FUNCTION "A-Outputs_valves" : Void
TITLE = Output_valves
{ S7_Optimized_Access := 'TRUE' }
AUTHOR : PiotrSlezak
FAMILY : Vorster
VERSION : 0.1
//Funkcja sterująca mechanizmami. Diagnostyka czujników, luzowanie, obsługa hamulca i wizualizacja stanów
   VAR_TEMP
      dummy : Bool;
      brake : Bool;
   END_VAR


BEGIN
NETWORK
TITLE = [1] GN BLOKADA_SRUBY_LEWY - HP
//[1] GN SCREW_LOCK_LEFT - HP
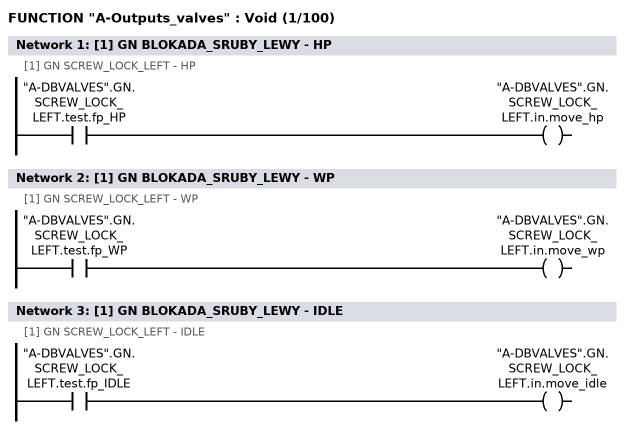
      O "A-DBVALVES".GN.SCREW_LOCK_LEFT.test.fp_HP;
//    O     "A-Flags".STATION.IN_HP_STEP
      = "A-DBVALVES".GN.SCREW_LOCK_LEFT.in.move_hp;
NETWORK
TITLE = [1] GN BLOKADA_SRUBY_LEWY - WP
//[1] GN SCREW_LOCK_LEFT - WP
      O "A-DBVALVES".GN.SCREW_LOCK_LEFT.test.fp_WP;
      = "A-DBVALVES".GN.SCREW_LOCK_LEFT.in.move_wp;
NETWORK
TITLE = [1] GN BLOKADA_SRUBY_LEWY - IDLE
//[1] GN SCREW_LOCK_LEFT - IDLE
      O "A-DBVALVES".GN.SCREW_LOCK_LEFT.test.fp_IDLE;
      = "A-DBVALVES".GN.SCREW_LOCK_LEFT.in.move_idle;
NETWORK
TITLE = [1] GN BLOKADA_SRUBY_LEWY
//[1] GN SCREW_LOCK_LEFT
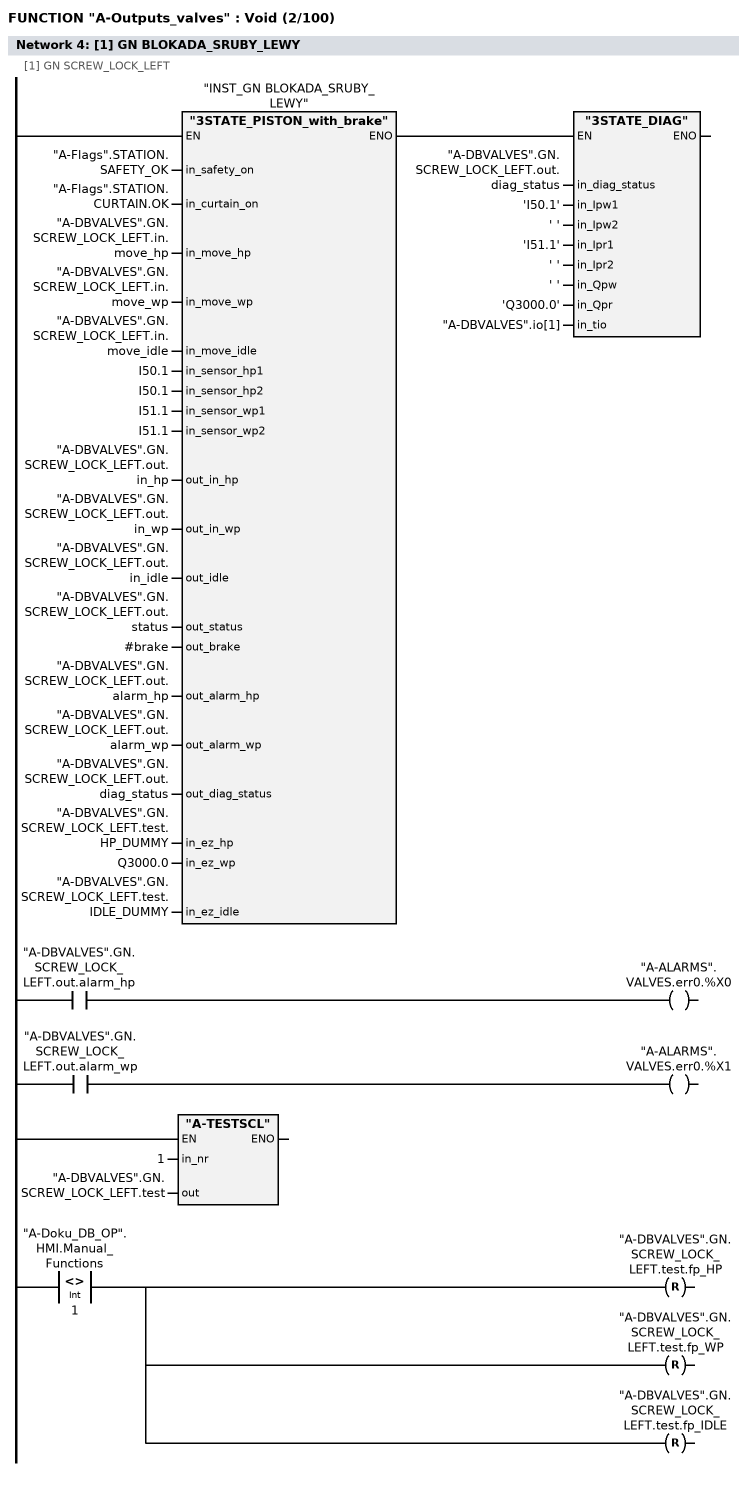
      CALL "3STATE_PISTON_with_brake", "INST_GN BLOKADA_SRUBY_LEWY"
      (  in_safety_on                := "A-Flags".STATION.SAFETY_OK ,
         in_curtain_on               := "A-Flags".STATION.CURTAIN.OK ,
         in_move_hp                  := "A-DBVALVES".GN.SCREW_LOCK_LEFT.in.move_hp ,
         in_move_wp                  := "A-DBVALVES".GN.SCREW_LOCK_LEFT.in.move_wp ,
         in_move_idle                := "A-DBVALVES".GN.SCREW_LOCK_LEFT.in.move_idle ,
         in_sensor_hp1               := I50.1 ,
         in_sensor_hp2               := I50.1 ,
         in_sensor_wp1               := I51.1 ,
         in_sensor_wp2               := I51.1 ,
         out_in_hp                   := "A-DBVALVES".GN.SCREW_LOCK_LEFT.out.in_hp ,
         out_in_wp                   := "A-DBVALVES".GN.SCREW_LOCK_LEFT.out.in_wp ,
         out_idle                    := "A-DBVALVES".GN.SCREW_LOCK_LEFT.out.in_idle ,
         out_status                  := "A-DBVALVES".GN.SCREW_LOCK_LEFT.out.status ,
         out_brake                   := #brake ,
         out_alarm_hp                := "A-DBVALVES".GN.SCREW_LOCK_LEFT.out.alarm_hp ,
         out_alarm_wp                := "A-DBVALVES".GN.SCREW_LOCK_LEFT.out.alarm_wp ,
         out_diag_status             := "A-DBVALVES".GN.SCREW_LOCK_LEFT.out.diag_status ,
         in_ez_hp                    := "A-DBVALVES".GN.SCREW_LOCK_LEFT.test.HP_DUMMY ,
         in_ez_wp                    := Q3000.0 ,
         in_ez_idle                  := "A-DBVALVES".GN.SCREW_LOCK_LEFT.test.IDLE_DUMMY
      );

      CALL "3STATE_DIAG"
      (  in_diag_status              := "A-DBVALVES".GN.SCREW_LOCK_LEFT.out.diag_status ,
         in_Ipw1                     := 'I50.1' ,
         in_Ipw2                     := ' ' ,
         in_Ipr1                     := 'I51.1' ,
         in_Ipr2                     := ' ' ,
         in_Qpw                      := ' ' ,
         in_Qpr                      := 'Q3000.0' ,
         in_tio                      := "A-DBVALVES".io[1]
      );

      A "A-DBVALVES".GN.SCREW_LOCK_LEFT.out.alarm_hp;
      = "A-ALARMS".VALVES.err0.%X0;

      A "A-DBVALVES".GN.SCREW_LOCK_LEFT.out.alarm_wp;
      = "A-ALARMS".VALVES.err0.%X1;

      CALL "A-TESTSCL"
      (  in_nr                       := 1 ,
         out                         := "A-DBVALVES".GN.SCREW_LOCK_LEFT.test
      );

      A(;
      L "A-Doku_DB_OP".HMI.Manual_Functions;
      L 1;
      <>I;
      );
      R "A-DBVALVES".GN.SCREW_LOCK_LEFT.test.fp_HP;
      R "A-DBVALVES".GN.SCREW_LOCK_LEFT.test.fp_WP;
      R "A-DBVALVES".GN.SCREW_LOCK_LEFT.test.fp_IDLE;
NETWORK
TITLE = -

NETWORK
TITLE = [2] GN BLOKADA_SRUBY_SRODEK - HP
//[2] GN SCREW_LOCK_MIDDLE - HP
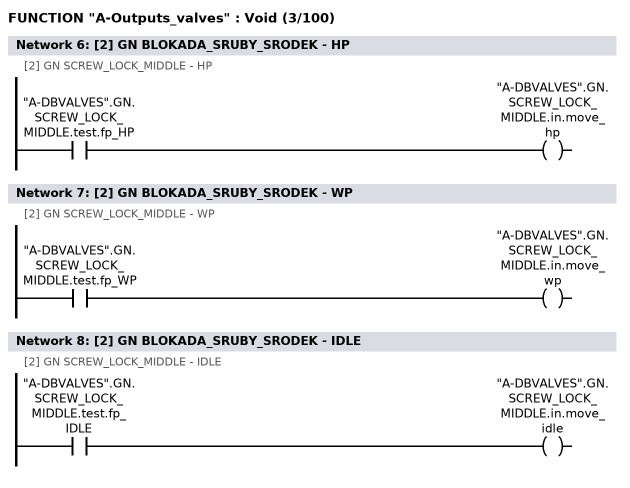
      O "A-DBVALVES".GN.SCREW_LOCK_MIDDLE.test.fp_HP;
//    O     "A-Flags".STATION.IN_HP_STEP
      = "A-DBVALVES".GN.SCREW_LOCK_MIDDLE.in.move_hp;
NETWORK
TITLE = [2] GN BLOKADA_SRUBY_SRODEK - WP
//[2] GN SCREW_LOCK_MIDDLE - WP
      O "A-DBVALVES".GN.SCREW_LOCK_MIDDLE.test.fp_WP;
      = "A-DBVALVES".GN.SCREW_LOCK_MIDDLE.in.move_wp;
NETWORK
TITLE = [2] GN BLOKADA_SRUBY_SRODEK - IDLE
//[2] GN SCREW_LOCK_MIDDLE - IDLE
      O "A-DBVALVES".GN.SCREW_LOCK_MIDDLE.test.fp_IDLE;
      = "A-DBVALVES".GN.SCREW_LOCK_MIDDLE.in.move_idle;
NETWORK
TITLE = [2] GN BLOKADA_SRUBY_SRODEK
//[2] GN SCREW_LOCK_MIDDLE
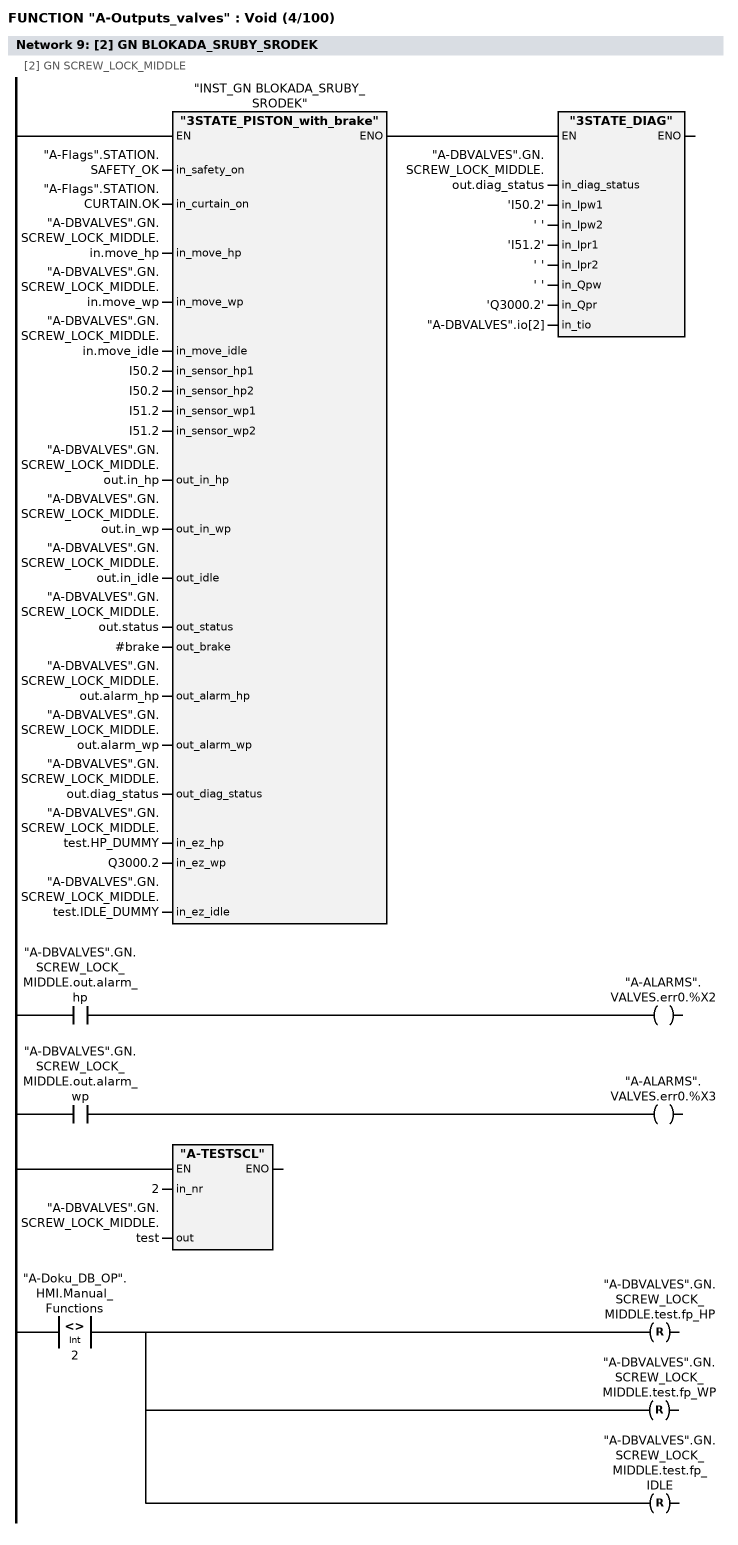
      CALL "3STATE_PISTON_with_brake", "INST_GN BLOKADA_SRUBY_SRODEK"
      (  in_safety_on                := "A-Flags".STATION.SAFETY_OK ,
         in_curtain_on               := "A-Flags".STATION.CURTAIN.OK ,
         in_move_hp                  := "A-DBVALVES".GN.SCREW_LOCK_MIDDLE.in.move_hp ,
         in_move_wp                  := "A-DBVALVES".GN.SCREW_LOCK_MIDDLE.in.move_wp ,
         in_move_idle                := "A-DBVALVES".GN.SCREW_LOCK_MIDDLE.in.move_idle ,
         in_sensor_hp1               := I50.2 ,
         in_sensor_hp2               := I50.2 ,
         in_sensor_wp1               := I51.2 ,
         in_sensor_wp2               := I51.2 ,
         out_in_hp                   := "A-DBVALVES".GN.SCREW_LOCK_MIDDLE.out.in_hp ,
         out_in_wp                   := "A-DBVALVES".GN.SCREW_LOCK_MIDDLE.out.in_wp ,
         out_idle                    := "A-DBVALVES".GN.SCREW_LOCK_MIDDLE.out.in_idle ,
         out_status                  := "A-DBVALVES".GN.SCREW_LOCK_MIDDLE.out.status ,
         out_brake                   := #brake ,
         out_alarm_hp                := "A-DBVALVES".GN.SCREW_LOCK_MIDDLE.out.alarm_hp ,
         out_alarm_wp                := "A-DBVALVES".GN.SCREW_LOCK_MIDDLE.out.alarm_wp ,
         out_diag_status             := "A-DBVALVES".GN.SCREW_LOCK_MIDDLE.out.diag_status ,
         in_ez_hp                    := "A-DBVALVES".GN.SCREW_LOCK_MIDDLE.test.HP_DUMMY ,
         in_ez_wp                    := Q3000.2 ,
         in_ez_idle                  := "A-DBVALVES".GN.SCREW_LOCK_MIDDLE.test.IDLE_DUMMY
      );

      CALL "3STATE_DIAG"
      (  in_diag_status              := "A-DBVALVES".GN.SCREW_LOCK_MIDDLE.out.diag_status ,
         in_Ipw1                     := 'I50.2' ,
         in_Ipw2                     := ' ' ,
         in_Ipr1                     := 'I51.2' ,
         in_Ipr2                     := ' ' ,
         in_Qpw                      := ' ' ,
         in_Qpr                      := 'Q3000.2' ,
         in_tio                      := "A-DBVALVES".io[2]
      );

      A "A-DBVALVES".GN.SCREW_LOCK_MIDDLE.out.alarm_hp;
      = "A-ALARMS".VALVES.err0.%X2;

      A "A-DBVALVES".GN.SCREW_LOCK_MIDDLE.out.alarm_wp;
      = "A-ALARMS".VALVES.err0.%X3;

      CALL "A-TESTSCL"
      (  in_nr                       := 2 ,
         out                         := "A-DBVALVES".GN.SCREW_LOCK_MIDDLE.test
      );

      A(;
      L "A-Doku_DB_OP".HMI.Manual_Functions;
      L 2;
      <>I;
      );
      R "A-DBVALVES".GN.SCREW_LOCK_MIDDLE.test.fp_HP;
      R "A-DBVALVES".GN.SCREW_LOCK_MIDDLE.test.fp_WP;
      R "A-DBVALVES".GN.SCREW_LOCK_MIDDLE.test.fp_IDLE;
NETWORK
TITLE = -

NETWORK
TITLE = [3] GN BLOKADA_SRUBY_PRAWY - HP
//[3] GN SCREW_LOCK_RIGHT - HP
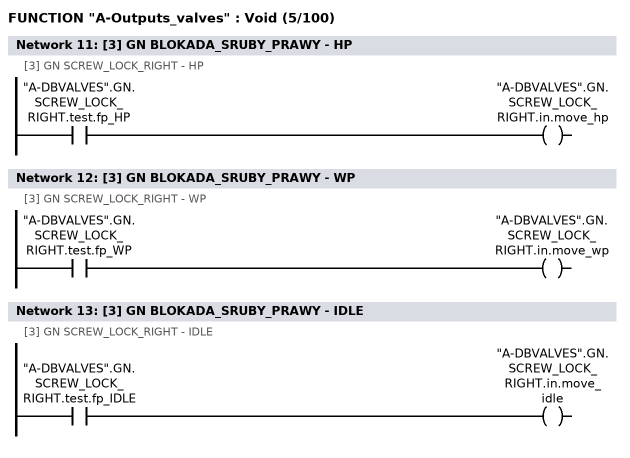
      O "A-DBVALVES".GN.SCREW_LOCK_RIGHT.test.fp_HP;
//    O     "A-Flags".STATION.IN_HP_STEP
      = "A-DBVALVES".GN.SCREW_LOCK_RIGHT.in.move_hp;
NETWORK
TITLE = [3] GN BLOKADA_SRUBY_PRAWY - WP
//[3] GN SCREW_LOCK_RIGHT - WP
      O "A-DBVALVES".GN.SCREW_LOCK_RIGHT.test.fp_WP;
      = "A-DBVALVES".GN.SCREW_LOCK_RIGHT.in.move_wp;
NETWORK
TITLE = [3] GN BLOKADA_SRUBY_PRAWY - IDLE
//[3] GN SCREW_LOCK_RIGHT - IDLE
      O "A-DBVALVES".GN.SCREW_LOCK_RIGHT.test.fp_IDLE;
      = "A-DBVALVES".GN.SCREW_LOCK_RIGHT.in.move_idle;
NETWORK
TITLE = [3] GN BLOKADA_SRUBY_PRAWY
//[3] GN SCREW_LOCK_RIGHT
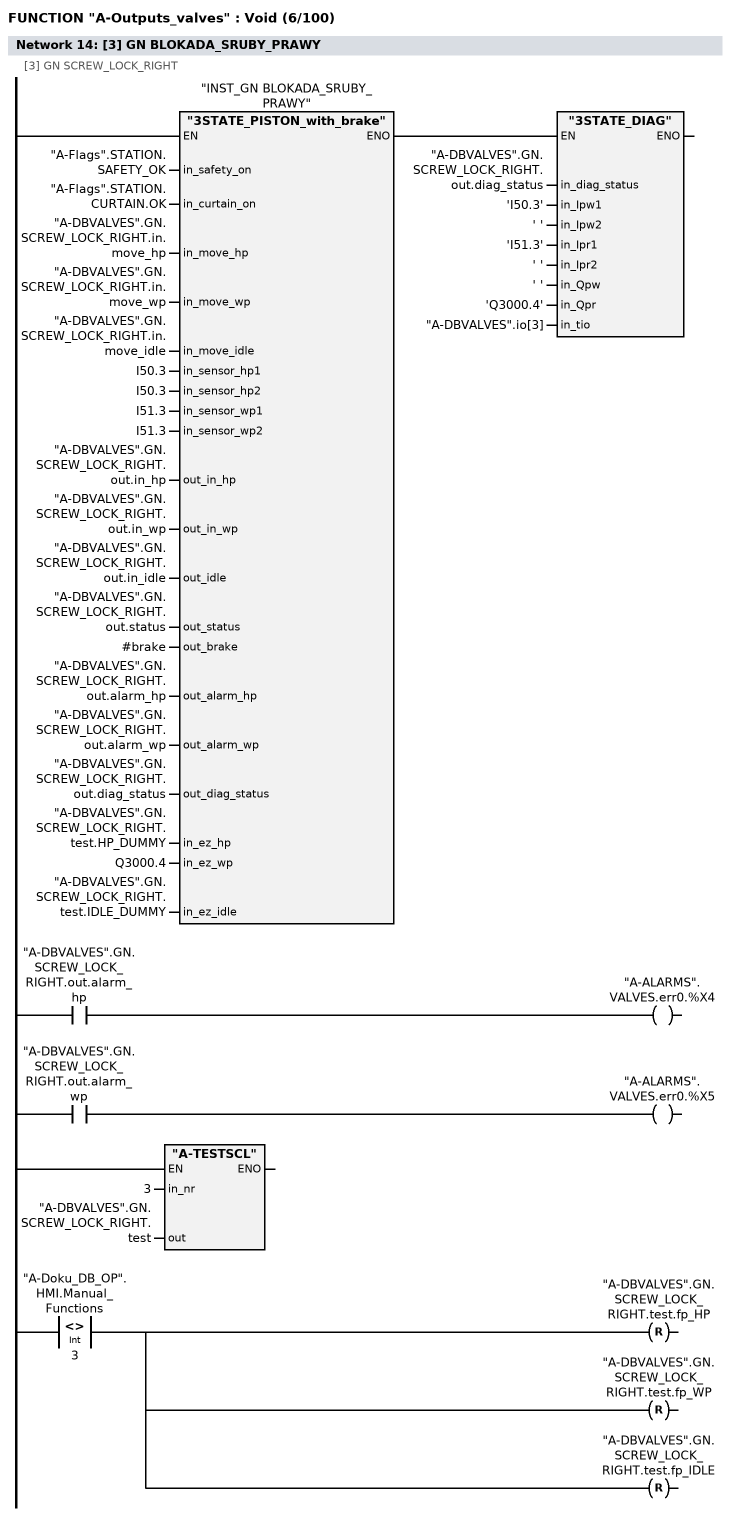
      CALL "3STATE_PISTON_with_brake", "INST_GN BLOKADA_SRUBY_PRAWY"
      (  in_safety_on                := "A-Flags".STATION.SAFETY_OK ,
         in_curtain_on               := "A-Flags".STATION.CURTAIN.OK ,
         in_move_hp                  := "A-DBVALVES".GN.SCREW_LOCK_RIGHT.in.move_hp ,
         in_move_wp                  := "A-DBVALVES".GN.SCREW_LOCK_RIGHT.in.move_wp ,
         in_move_idle                := "A-DBVALVES".GN.SCREW_LOCK_RIGHT.in.move_idle ,
         in_sensor_hp1               := I50.3 ,
         in_sensor_hp2               := I50.3 ,
         in_sensor_wp1               := I51.3 ,
         in_sensor_wp2               := I51.3 ,
         out_in_hp                   := "A-DBVALVES".GN.SCREW_LOCK_RIGHT.out.in_hp ,
         out_in_wp                   := "A-DBVALVES".GN.SCREW_LOCK_RIGHT.out.in_wp ,
         out_idle                    := "A-DBVALVES".GN.SCREW_LOCK_RIGHT.out.in_idle ,
         out_status                  := "A-DBVALVES".GN.SCREW_LOCK_RIGHT.out.status ,
         out_brake                   := #brake ,
         out_alarm_hp                := "A-DBVALVES".GN.SCREW_LOCK_RIGHT.out.alarm_hp ,
         out_alarm_wp                := "A-DBVALVES".GN.SCREW_LOCK_RIGHT.out.alarm_wp ,
         out_diag_status             := "A-DBVALVES".GN.SCREW_LOCK_RIGHT.out.diag_status ,
         in_ez_hp                    := "A-DBVALVES".GN.SCREW_LOCK_RIGHT.test.HP_DUMMY ,
         in_ez_wp                    := Q3000.4 ,
         in_ez_idle                  := "A-DBVALVES".GN.SCREW_LOCK_RIGHT.test.IDLE_DUMMY
      );

      CALL "3STATE_DIAG"
      (  in_diag_status              := "A-DBVALVES".GN.SCREW_LOCK_RIGHT.out.diag_status ,
         in_Ipw1                     := 'I50.3' ,
         in_Ipw2                     := ' ' ,
         in_Ipr1                     := 'I51.3' ,
         in_Ipr2                     := ' ' ,
         in_Qpw                      := ' ' ,
         in_Qpr                      := 'Q3000.4' ,
         in_tio                      := "A-DBVALVES".io[3]
      );

      A "A-DBVALVES".GN.SCREW_LOCK_RIGHT.out.alarm_hp;
      = "A-ALARMS".VALVES.err0.%X4;

      A "A-DBVALVES".GN.SCREW_LOCK_RIGHT.out.alarm_wp;
      = "A-ALARMS".VALVES.err0.%X5;

      CALL "A-TESTSCL"
      (  in_nr                       := 3 ,
         out                         := "A-DBVALVES".GN.SCREW_LOCK_RIGHT.test
      );

      A(;
      L "A-Doku_DB_OP".HMI.Manual_Functions;
      L 3;
      <>I;
      );
      R "A-DBVALVES".GN.SCREW_LOCK_RIGHT.test.fp_HP;
      R "A-DBVALVES".GN.SCREW_LOCK_RIGHT.test.fp_WP;
      R "A-DBVALVES".GN.SCREW_LOCK_RIGHT.test.fp_IDLE;
NETWORK
TITLE = -

NETWORK
TITLE = [4] GN ZASUWKA - HP
//[4] GN LATCH - HP
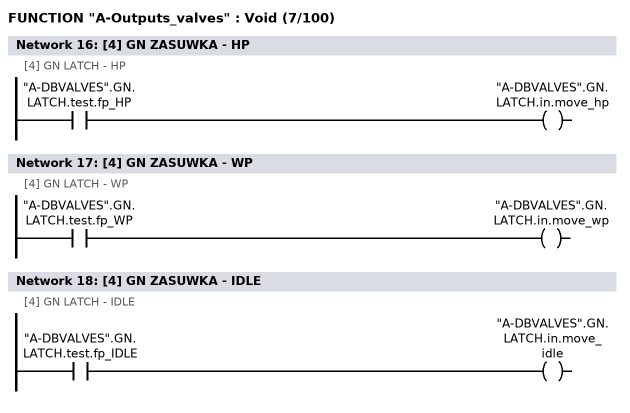
      O "A-DBVALVES".GN.LATCH.test.fp_HP;
//    O     "A-Flags".STATION.IN_HP_STEP
      = "A-DBVALVES".GN.LATCH.in.move_hp;
NETWORK
TITLE = [4] GN ZASUWKA - WP
//[4] GN LATCH - WP
      O "A-DBVALVES".GN.LATCH.test.fp_WP;
      = "A-DBVALVES".GN.LATCH.in.move_wp;
NETWORK
TITLE = [4] GN ZASUWKA - IDLE
//[4] GN LATCH - IDLE
      O "A-DBVALVES".GN.LATCH.test.fp_IDLE;
      = "A-DBVALVES".GN.LATCH.in.move_idle;
NETWORK
TITLE = [4] GN ZASUWKA
//[4] GN LATCH
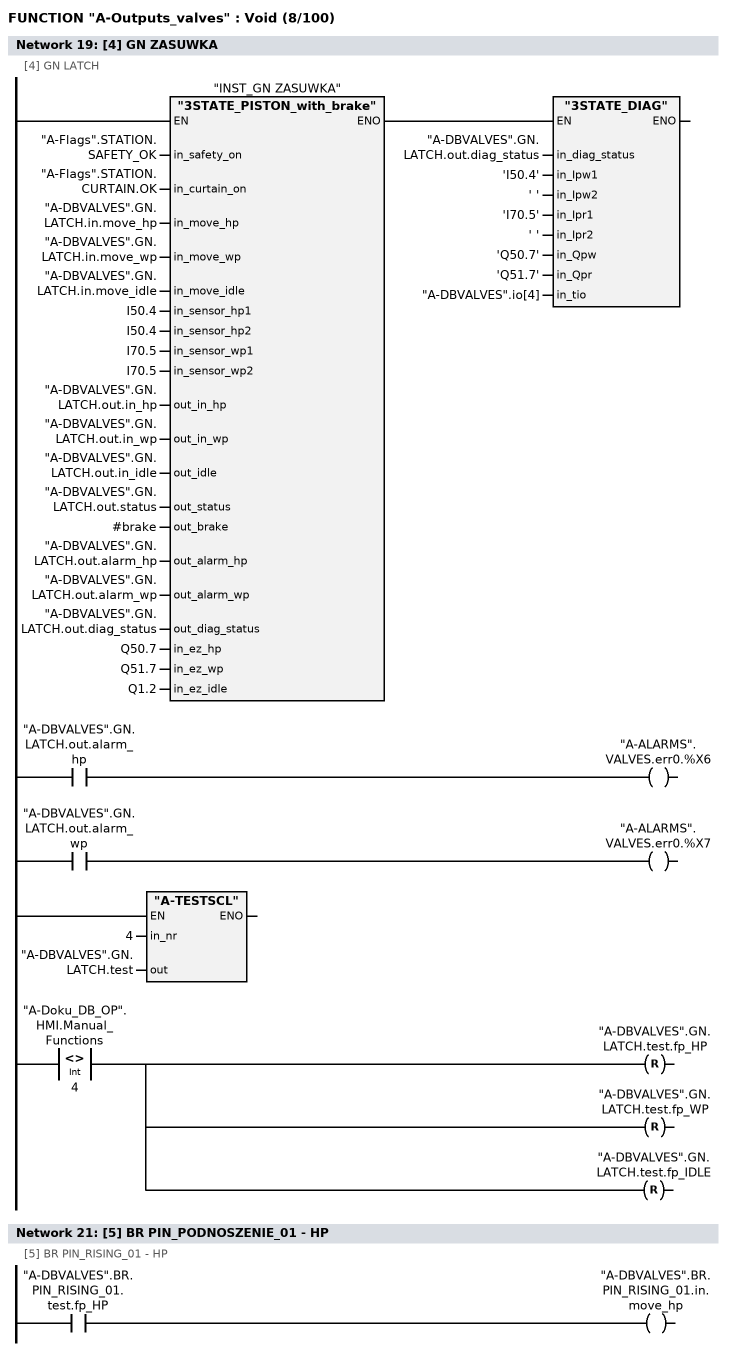
      CALL "3STATE_PISTON_with_brake", "INST_GN ZASUWKA"
      (  in_safety_on                := "A-Flags".STATION.SAFETY_OK ,
         in_curtain_on               := "A-Flags".STATION.CURTAIN.OK ,
         in_move_hp                  := "A-DBVALVES".GN.LATCH.in.move_hp ,
         in_move_wp                  := "A-DBVALVES".GN.LATCH.in.move_wp ,
         in_move_idle                := "A-DBVALVES".GN.LATCH.in.move_idle ,
         in_sensor_hp1               := I50.4 ,
         in_sensor_hp2               := I50.4 ,
         in_sensor_wp1               := I70.5 ,
         in_sensor_wp2               := I70.5 ,
         out_in_hp                   := "A-DBVALVES".GN.LATCH.out.in_hp ,
         out_in_wp                   := "A-DBVALVES".GN.LATCH.out.in_wp ,
         out_idle                    := "A-DBVALVES".GN.LATCH.out.in_idle ,
         out_status                  := "A-DBVALVES".GN.LATCH.out.status ,
         out_brake                   := #brake ,
         out_alarm_hp                := "A-DBVALVES".GN.LATCH.out.alarm_hp ,
         out_alarm_wp                := "A-DBVALVES".GN.LATCH.out.alarm_wp ,
         out_diag_status             := "A-DBVALVES".GN.LATCH.out.diag_status ,
         in_ez_hp                    := Q50.7 ,
         in_ez_wp                    := Q51.7 ,
         in_ez_idle                  := Q1.2
      );

      CALL "3STATE_DIAG"
      (  in_diag_status              := "A-DBVALVES".GN.LATCH.out.diag_status ,
         in_Ipw1                     := 'I50.4' ,
         in_Ipw2                     := ' ' ,
         in_Ipr1                     := 'I70.5' ,
         in_Ipr2                     := ' ' ,
         in_Qpw                      := 'Q50.7' ,
         in_Qpr                      := 'Q51.7' ,
         in_tio                      := "A-DBVALVES".io[4]
      );

      A "A-DBVALVES".GN.LATCH.out.alarm_hp;
      = "A-ALARMS".VALVES.err0.%X6;

      A "A-DBVALVES".GN.LATCH.out.alarm_wp;
      = "A-ALARMS".VALVES.err0.%X7;

      CALL "A-TESTSCL"
      (  in_nr                       := 4 ,
         out                         := "A-DBVALVES".GN.LATCH.test
      );

      A(;
      L "A-Doku_DB_OP".HMI.Manual_Functions;
      L 4;
      <>I;
      );
      R "A-DBVALVES".GN.LATCH.test.fp_HP;
      R "A-DBVALVES".GN.LATCH.test.fp_WP;
      R "A-DBVALVES".GN.LATCH.test.fp_IDLE;
NETWORK
TITLE = -

NETWORK
TITLE = [5] BR PIN_PODNOSZENIE_01 - HP
//[5] BR PIN_RISING_01 - HP
      O "A-DBVALVES".BR.PIN_RISING_01.test.fp_HP;
//    O     "A-Flags".STATION.IN_HP_STEP
      = "A-DBVALVES".BR.PIN_RISING_01.in.move_hp;
NETWORK
TITLE = [5] BR PIN_PODNOSZENIE_01 - WP
//[5] BR PIN_RISING_01 - WP
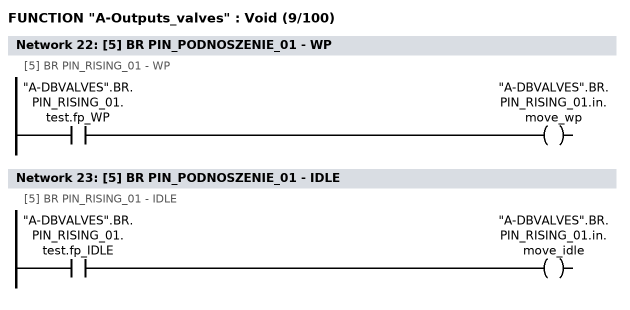
      O "A-DBVALVES".BR.PIN_RISING_01.test.fp_WP;
      = "A-DBVALVES".BR.PIN_RISING_01.in.move_wp;
NETWORK
TITLE = [5] BR PIN_PODNOSZENIE_01 - IDLE
//[5] BR PIN_RISING_01 - IDLE
      O "A-DBVALVES".BR.PIN_RISING_01.test.fp_IDLE;
      = "A-DBVALVES".BR.PIN_RISING_01.in.move_idle;
NETWORK
TITLE = [5] BR PIN_PODNOSZENIE_01
//[5] BR PIN_RISING_01
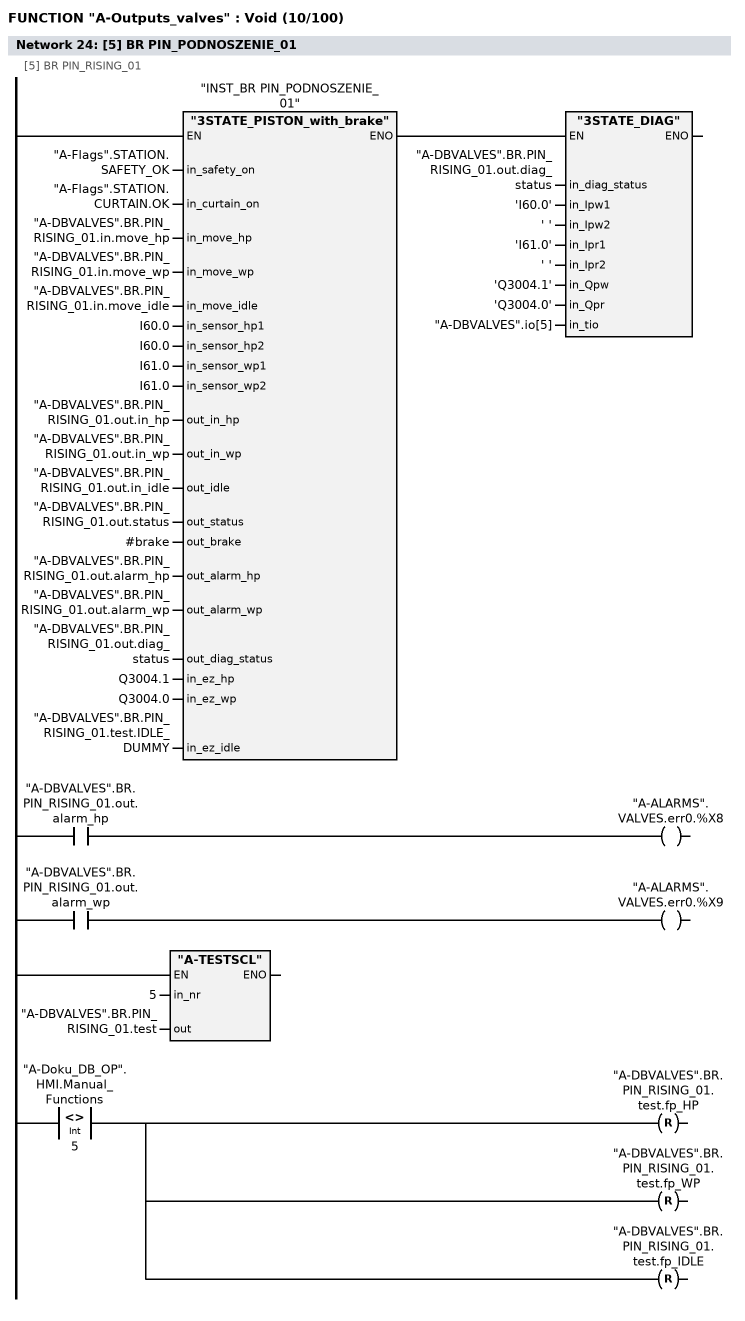
      CALL "3STATE_PISTON_with_brake", "INST_BR PIN_PODNOSZENIE_01"
      (  in_safety_on                := "A-Flags".STATION.SAFETY_OK ,
         in_curtain_on               := "A-Flags".STATION.CURTAIN.OK ,
         in_move_hp                  := "A-DBVALVES".BR.PIN_RISING_01.in.move_hp ,
         in_move_wp                  := "A-DBVALVES".BR.PIN_RISING_01.in.move_wp ,
         in_move_idle                := "A-DBVALVES".BR.PIN_RISING_01.in.move_idle ,
         in_sensor_hp1               := I60.0 ,
         in_sensor_hp2               := I60.0 ,
         in_sensor_wp1               := I61.0 ,
         in_sensor_wp2               := I61.0 ,
         out_in_hp                   := "A-DBVALVES".BR.PIN_RISING_01.out.in_hp ,
         out_in_wp                   := "A-DBVALVES".BR.PIN_RISING_01.out.in_wp ,
         out_idle                    := "A-DBVALVES".BR.PIN_RISING_01.out.in_idle ,
         out_status                  := "A-DBVALVES".BR.PIN_RISING_01.out.status ,
         out_brake                   := #brake ,
         out_alarm_hp                := "A-DBVALVES".BR.PIN_RISING_01.out.alarm_hp ,
         out_alarm_wp                := "A-DBVALVES".BR.PIN_RISING_01.out.alarm_wp ,
         out_diag_status             := "A-DBVALVES".BR.PIN_RISING_01.out.diag_status ,
         in_ez_hp                    := Q3004.1 ,
         in_ez_wp                    := Q3004.0 ,
         in_ez_idle                  := "A-DBVALVES".BR.PIN_RISING_01.test.IDLE_DUMMY
      );

      CALL "3STATE_DIAG"
      (  in_diag_status              := "A-DBVALVES".BR.PIN_RISING_01.out.diag_status ,
         in_Ipw1                     := 'I60.0' ,
         in_Ipw2                     := ' ' ,
         in_Ipr1                     := 'I61.0' ,
         in_Ipr2                     := ' ' ,
         in_Qpw                      := 'Q3004.1' ,
         in_Qpr                      := 'Q3004.0' ,
         in_tio                      := "A-DBVALVES".io[5]
      );

      A "A-DBVALVES".BR.PIN_RISING_01.out.alarm_hp;
      = "A-ALARMS".VALVES.err0.%X8;

      A "A-DBVALVES".BR.PIN_RISING_01.out.alarm_wp;
      = "A-ALARMS".VALVES.err0.%X9;

      CALL "A-TESTSCL"
      (  in_nr                       := 5 ,
         out                         := "A-DBVALVES".BR.PIN_RISING_01.test
      );

      A(;
      L "A-Doku_DB_OP".HMI.Manual_Functions;
      L 5;
      <>I;
      );
      R "A-DBVALVES".BR.PIN_RISING_01.test.fp_HP;
      R "A-DBVALVES".BR.PIN_RISING_01.test.fp_WP;
      R "A-DBVALVES".BR.PIN_RISING_01.test.fp_IDLE;
NETWORK
TITLE = -

NETWORK
TITLE = [6] BR PIN_01 - HP
//[6] BR PIN_01 - HP
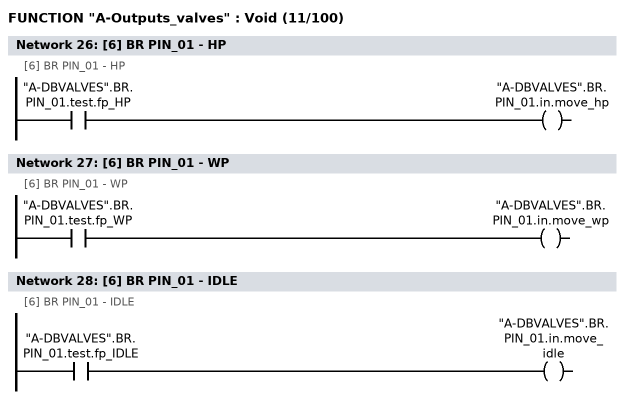
      O "A-DBVALVES".BR.PIN_01.test.fp_HP;
//    O     "A-Flags".STATION.IN_HP_STEP
      = "A-DBVALVES".BR.PIN_01.in.move_hp;
NETWORK
TITLE = [6] BR PIN_01 - WP
//[6] BR PIN_01 - WP
      O "A-DBVALVES".BR.PIN_01.test.fp_WP;
      = "A-DBVALVES".BR.PIN_01.in.move_wp;
NETWORK
TITLE = [6] BR PIN_01 - IDLE
//[6] BR PIN_01 - IDLE
      O "A-DBVALVES".BR.PIN_01.test.fp_IDLE;
      = "A-DBVALVES".BR.PIN_01.in.move_idle;
NETWORK
TITLE = [6] BR PIN_01
//[6] BR PIN_01
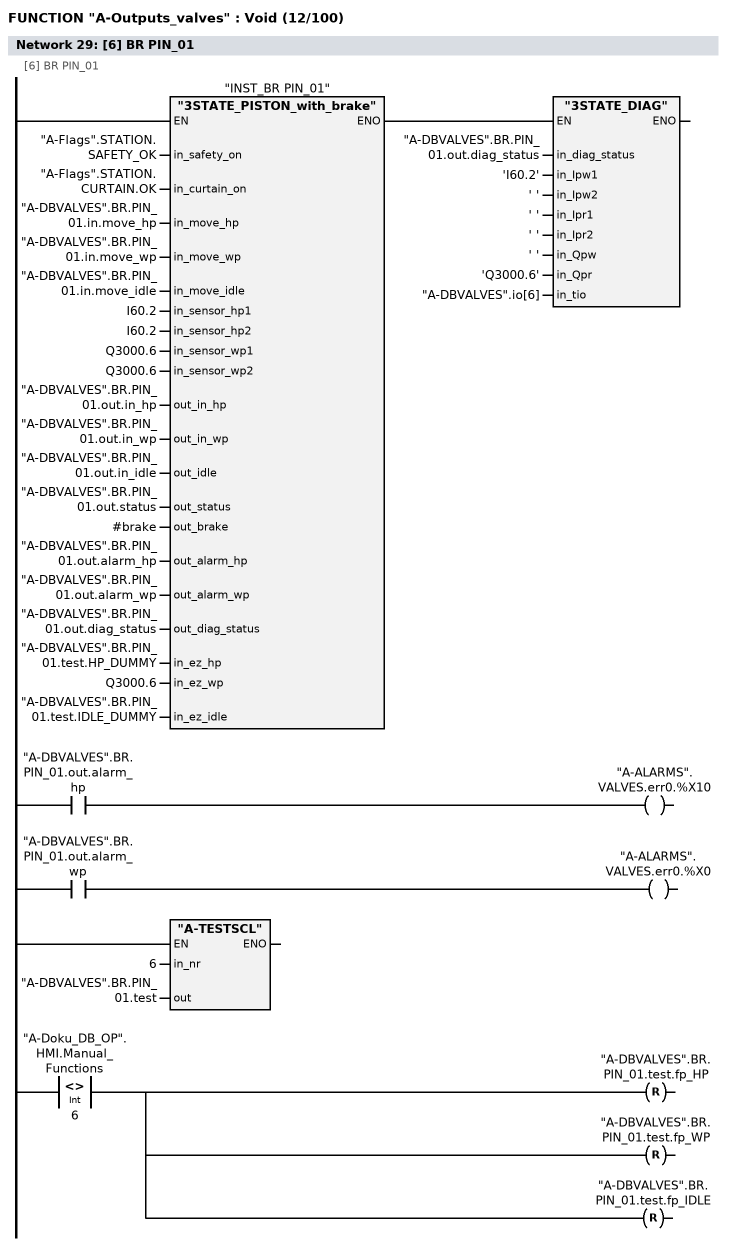
      CALL "3STATE_PISTON_with_brake", "INST_BR PIN_01"
      (  in_safety_on                := "A-Flags".STATION.SAFETY_OK ,
         in_curtain_on               := "A-Flags".STATION.CURTAIN.OK ,
         in_move_hp                  := "A-DBVALVES".BR.PIN_01.in.move_hp ,
         in_move_wp                  := "A-DBVALVES".BR.PIN_01.in.move_wp ,
         in_move_idle                := "A-DBVALVES".BR.PIN_01.in.move_idle ,
         in_sensor_hp1               := I60.2 ,
         in_sensor_hp2               := I60.2 ,
         in_sensor_wp1               := Q3000.6 ,
         in_sensor_wp2               := Q3000.6 ,
         out_in_hp                   := "A-DBVALVES".BR.PIN_01.out.in_hp ,
         out_in_wp                   := "A-DBVALVES".BR.PIN_01.out.in_wp ,
         out_idle                    := "A-DBVALVES".BR.PIN_01.out.in_idle ,
         out_status                  := "A-DBVALVES".BR.PIN_01.out.status ,
         out_brake                   := #brake ,
         out_alarm_hp                := "A-DBVALVES".BR.PIN_01.out.alarm_hp ,
         out_alarm_wp                := "A-DBVALVES".BR.PIN_01.out.alarm_wp ,
         out_diag_status             := "A-DBVALVES".BR.PIN_01.out.diag_status ,
         in_ez_hp                    := "A-DBVALVES".BR.PIN_01.test.HP_DUMMY ,
         in_ez_wp                    := Q3000.6 ,
         in_ez_idle                  := "A-DBVALVES".BR.PIN_01.test.IDLE_DUMMY
      );

      CALL "3STATE_DIAG"
      (  in_diag_status              := "A-DBVALVES".BR.PIN_01.out.diag_status ,
         in_Ipw1                     := 'I60.2' ,
         in_Ipw2                     := ' ' ,
         in_Ipr1                     := ' ' ,
         in_Ipr2                     := ' ' ,
         in_Qpw                      := ' ' ,
         in_Qpr                      := 'Q3000.6' ,
         in_tio                      := "A-DBVALVES".io[6]
      );

      A "A-DBVALVES".BR.PIN_01.out.alarm_hp;
      = "A-ALARMS".VALVES.err0.%X10;

      A "A-DBVALVES".BR.PIN_01.out.alarm_wp;
      = "A-ALARMS".VALVES.err0.%X0;

      CALL "A-TESTSCL"
      (  in_nr                       := 6 ,
         out                         := "A-DBVALVES".BR.PIN_01.test
      );

      A(;
      L "A-Doku_DB_OP".HMI.Manual_Functions;
      L 6;
      <>I;
      );
      R "A-DBVALVES".BR.PIN_01.test.fp_HP;
      R "A-DBVALVES".BR.PIN_01.test.fp_WP;
      R "A-DBVALVES".BR.PIN_01.test.fp_IDLE;
NETWORK
TITLE = -

NETWORK
TITLE = [7] BR PIN_PODNOSZENIE_02 - HP
//[7] BR PIN_RISING_02 - HP
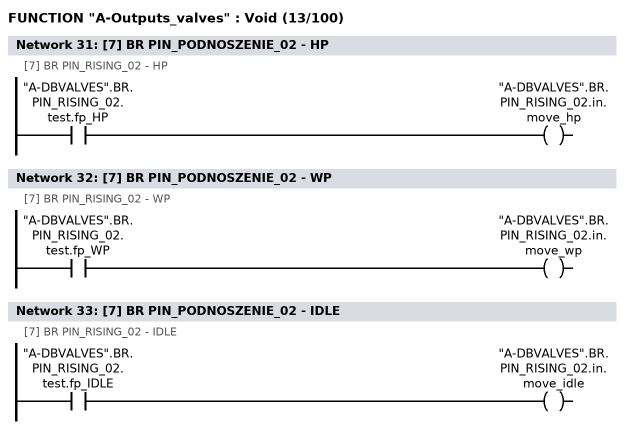
      O "A-DBVALVES".BR.PIN_RISING_02.test.fp_HP;
//    O     "A-Flags".STATION.IN_HP_STEP
      = "A-DBVALVES".BR.PIN_RISING_02.in.move_hp;
NETWORK
TITLE = [7] BR PIN_PODNOSZENIE_02 - WP
//[7] BR PIN_RISING_02 - WP
      O "A-DBVALVES".BR.PIN_RISING_02.test.fp_WP;
      = "A-DBVALVES".BR.PIN_RISING_02.in.move_wp;
NETWORK
TITLE = [7] BR PIN_PODNOSZENIE_02 - IDLE
//[7] BR PIN_RISING_02 - IDLE
      O "A-DBVALVES".BR.PIN_RISING_02.test.fp_IDLE;
      = "A-DBVALVES".BR.PIN_RISING_02.in.move_idle;
NETWORK
TITLE = [7] BR PIN_PODNOSZENIE_02
//[7] BR PIN_RISING_02
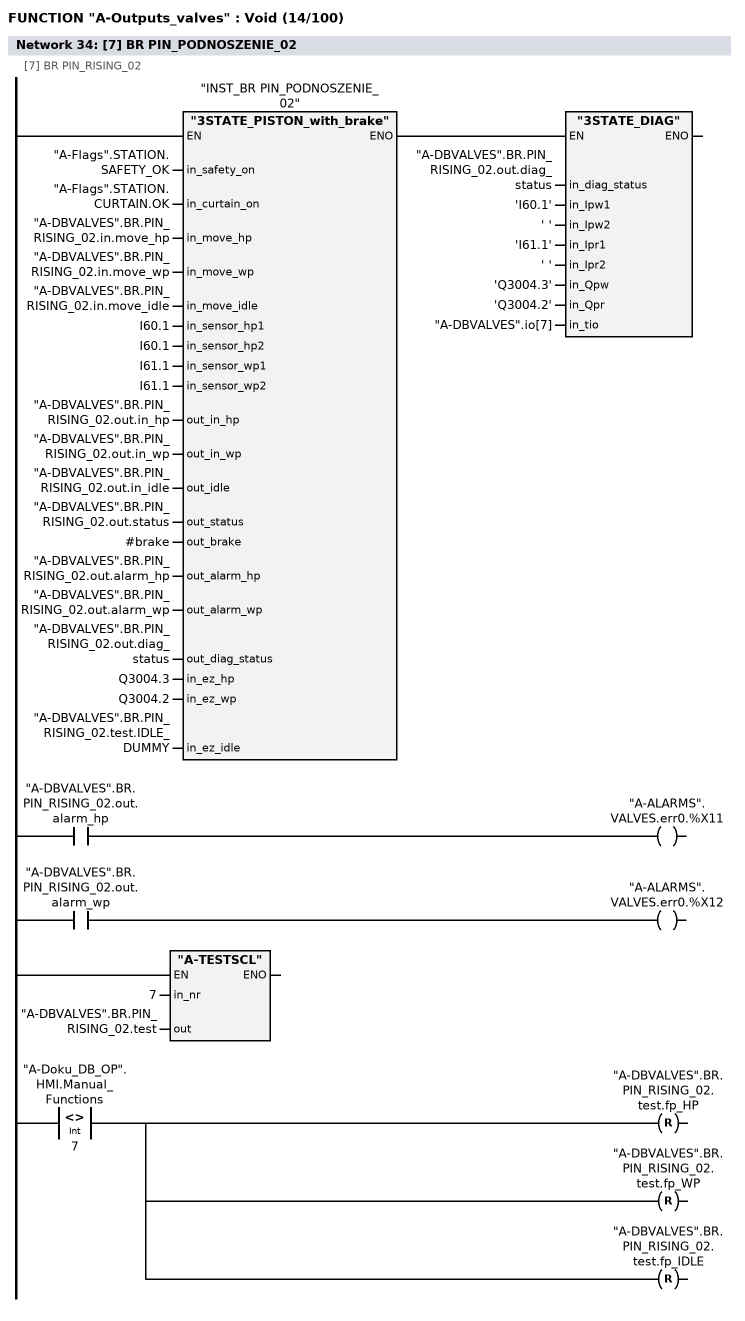
      CALL "3STATE_PISTON_with_brake", "INST_BR PIN_PODNOSZENIE_02"
      (  in_safety_on                := "A-Flags".STATION.SAFETY_OK ,
         in_curtain_on               := "A-Flags".STATION.CURTAIN.OK ,
         in_move_hp                  := "A-DBVALVES".BR.PIN_RISING_02.in.move_hp ,
         in_move_wp                  := "A-DBVALVES".BR.PIN_RISING_02.in.move_wp ,
         in_move_idle                := "A-DBVALVES".BR.PIN_RISING_02.in.move_idle ,
         in_sensor_hp1               := I60.1 ,
         in_sensor_hp2               := I60.1 ,
         in_sensor_wp1               := I61.1 ,
         in_sensor_wp2               := I61.1 ,
         out_in_hp                   := "A-DBVALVES".BR.PIN_RISING_02.out.in_hp ,
         out_in_wp                   := "A-DBVALVES".BR.PIN_RISING_02.out.in_wp ,
         out_idle                    := "A-DBVALVES".BR.PIN_RISING_02.out.in_idle ,
         out_status                  := "A-DBVALVES".BR.PIN_RISING_02.out.status ,
         out_brake                   := #brake ,
         out_alarm_hp                := "A-DBVALVES".BR.PIN_RISING_02.out.alarm_hp ,
         out_alarm_wp                := "A-DBVALVES".BR.PIN_RISING_02.out.alarm_wp ,
         out_diag_status             := "A-DBVALVES".BR.PIN_RISING_02.out.diag_status ,
         in_ez_hp                    := Q3004.3 ,
         in_ez_wp                    := Q3004.2 ,
         in_ez_idle                  := "A-DBVALVES".BR.PIN_RISING_02.test.IDLE_DUMMY
      );

      CALL "3STATE_DIAG"
      (  in_diag_status              := "A-DBVALVES".BR.PIN_RISING_02.out.diag_status ,
         in_Ipw1                     := 'I60.1' ,
         in_Ipw2                     := ' ' ,
         in_Ipr1                     := 'I61.1' ,
         in_Ipr2                     := ' ' ,
         in_Qpw                      := 'Q3004.3' ,
         in_Qpr                      := 'Q3004.2' ,
         in_tio                      := "A-DBVALVES".io[7]
      );

      A "A-DBVALVES".BR.PIN_RISING_02.out.alarm_hp;
      = "A-ALARMS".VALVES.err0.%X11;

      A "A-DBVALVES".BR.PIN_RISING_02.out.alarm_wp;
      = "A-ALARMS".VALVES.err0.%X12;

      CALL "A-TESTSCL"
      (  in_nr                       := 7 ,
         out                         := "A-DBVALVES".BR.PIN_RISING_02.test
      );

      A(;
      L "A-Doku_DB_OP".HMI.Manual_Functions;
      L 7;
      <>I;
      );
      R "A-DBVALVES".BR.PIN_RISING_02.test.fp_HP;
      R "A-DBVALVES".BR.PIN_RISING_02.test.fp_WP;
      R "A-DBVALVES".BR.PIN_RISING_02.test.fp_IDLE;
NETWORK
TITLE = -

NETWORK
TITLE = [8] BR PIN_02 - HP
//[8] BR PIN_02 - HP
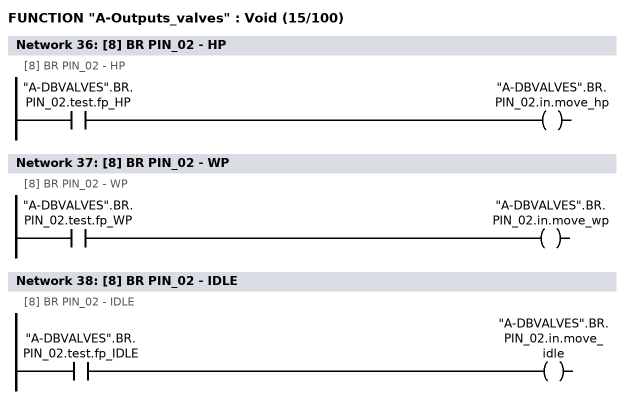
      O "A-DBVALVES".BR.PIN_02.test.fp_HP;
//    O     "A-Flags".STATION.IN_HP_STEP
      = "A-DBVALVES".BR.PIN_02.in.move_hp;
NETWORK
TITLE = [8] BR PIN_02 - WP
//[8] BR PIN_02 - WP
      O "A-DBVALVES".BR.PIN_02.test.fp_WP;
      = "A-DBVALVES".BR.PIN_02.in.move_wp;
NETWORK
TITLE = [8] BR PIN_02 - IDLE
//[8] BR PIN_02 - IDLE
      O "A-DBVALVES".BR.PIN_02.test.fp_IDLE;
      = "A-DBVALVES".BR.PIN_02.in.move_idle;
NETWORK
TITLE = [8] BR PIN_02
//[8] BR PIN_02
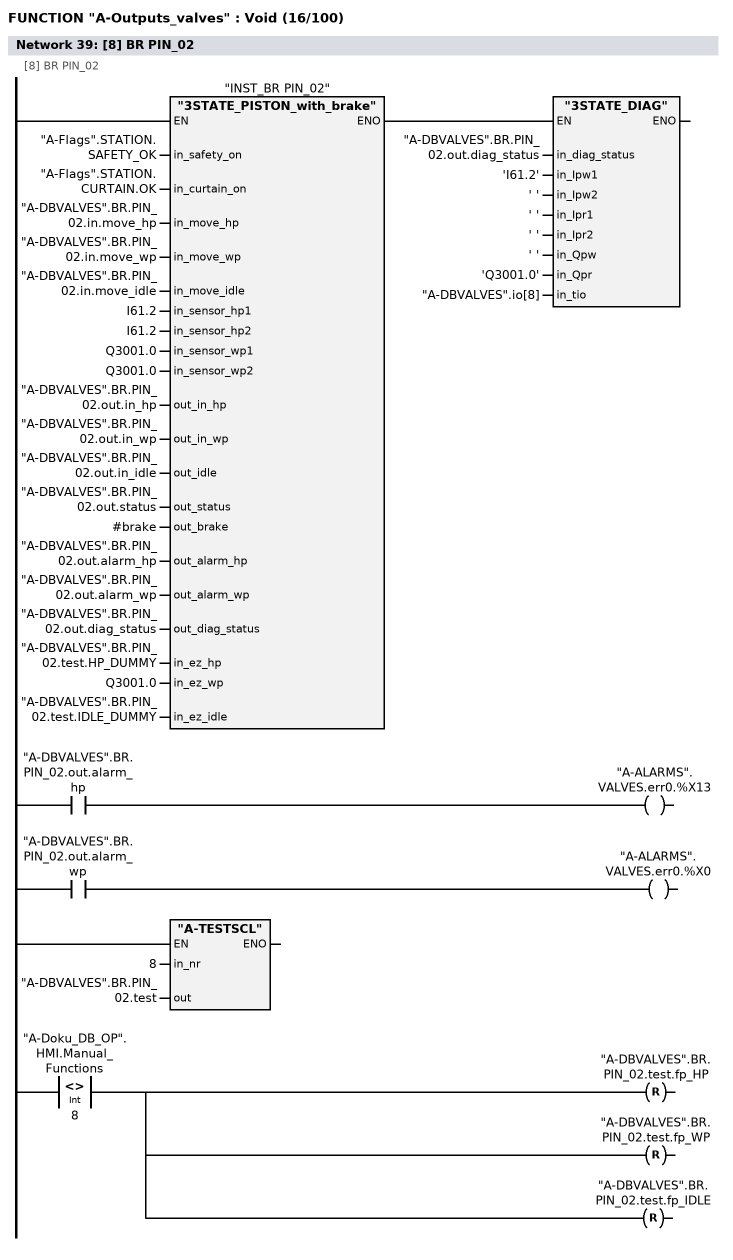
      CALL "3STATE_PISTON_with_brake", "INST_BR PIN_02"
      (  in_safety_on                := "A-Flags".STATION.SAFETY_OK ,
         in_curtain_on               := "A-Flags".STATION.CURTAIN.OK ,
         in_move_hp                  := "A-DBVALVES".BR.PIN_02.in.move_hp ,
         in_move_wp                  := "A-DBVALVES".BR.PIN_02.in.move_wp ,
         in_move_idle                := "A-DBVALVES".BR.PIN_02.in.move_idle ,
         in_sensor_hp1               := I61.2 ,
         in_sensor_hp2               := I61.2 ,
         in_sensor_wp1               := Q3001.0 ,
         in_sensor_wp2               := Q3001.0 ,
         out_in_hp                   := "A-DBVALVES".BR.PIN_02.out.in_hp ,
         out_in_wp                   := "A-DBVALVES".BR.PIN_02.out.in_wp ,
         out_idle                    := "A-DBVALVES".BR.PIN_02.out.in_idle ,
         out_status                  := "A-DBVALVES".BR.PIN_02.out.status ,
         out_brake                   := #brake ,
         out_alarm_hp                := "A-DBVALVES".BR.PIN_02.out.alarm_hp ,
         out_alarm_wp                := "A-DBVALVES".BR.PIN_02.out.alarm_wp ,
         out_diag_status             := "A-DBVALVES".BR.PIN_02.out.diag_status ,
         in_ez_hp                    := "A-DBVALVES".BR.PIN_02.test.HP_DUMMY ,
         in_ez_wp                    := Q3001.0 ,
         in_ez_idle                  := "A-DBVALVES".BR.PIN_02.test.IDLE_DUMMY
      );

      CALL "3STATE_DIAG"
      (  in_diag_status              := "A-DBVALVES".BR.PIN_02.out.diag_status ,
         in_Ipw1                     := 'I61.2' ,
         in_Ipw2                     := ' ' ,
         in_Ipr1                     := ' ' ,
         in_Ipr2                     := ' ' ,
         in_Qpw                      := ' ' ,
         in_Qpr                      := 'Q3001.0' ,
         in_tio                      := "A-DBVALVES".io[8]
      );

      A "A-DBVALVES".BR.PIN_02.out.alarm_hp;
      = "A-ALARMS".VALVES.err0.%X13;

      A "A-DBVALVES".BR.PIN_02.out.alarm_wp;
      = "A-ALARMS".VALVES.err0.%X0;

      CALL "A-TESTSCL"
      (  in_nr                       := 8 ,
         out                         := "A-DBVALVES".BR.PIN_02.test
      );

      A(;
      L "A-Doku_DB_OP".HMI.Manual_Functions;
      L 8;
      <>I;
      );
      R "A-DBVALVES".BR.PIN_02.test.fp_HP;
      R "A-DBVALVES".BR.PIN_02.test.fp_WP;
      R "A-DBVALVES".BR.PIN_02.test.fp_IDLE;
NETWORK
TITLE = -

NETWORK
TITLE = [9] BR PIN_PODNOSZENIE_03 - HP
//[9] BR PIN_RISING_03 - HP
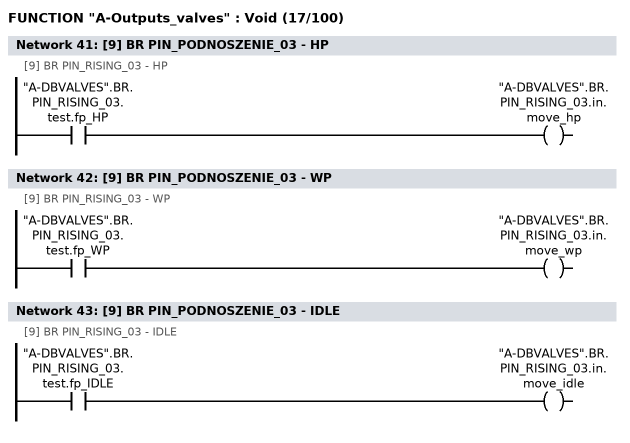
      O "A-DBVALVES".BR.PIN_RISING_03.test.fp_HP;
//    O     "A-Flags".STATION.IN_HP_STEP
      = "A-DBVALVES".BR.PIN_RISING_03.in.move_hp;
NETWORK
TITLE = [9] BR PIN_PODNOSZENIE_03 - WP
//[9] BR PIN_RISING_03 - WP
      O "A-DBVALVES".BR.PIN_RISING_03.test.fp_WP;
      = "A-DBVALVES".BR.PIN_RISING_03.in.move_wp;
NETWORK
TITLE = [9] BR PIN_PODNOSZENIE_03 - IDLE
//[9] BR PIN_RISING_03 - IDLE
      O "A-DBVALVES".BR.PIN_RISING_03.test.fp_IDLE;
      = "A-DBVALVES".BR.PIN_RISING_03.in.move_idle;
NETWORK
TITLE = [9] BR PIN_PODNOSZENIE_03
//[9] BR PIN_RISING_03
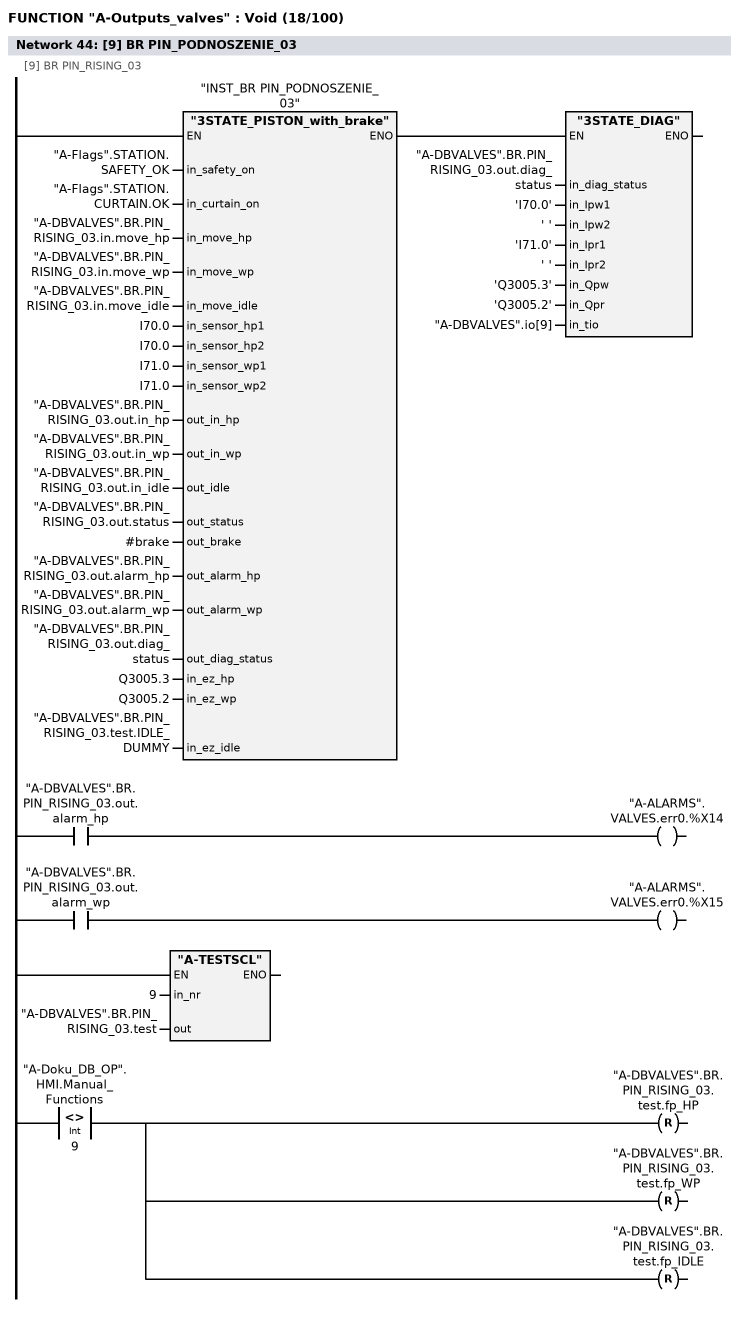
      CALL "3STATE_PISTON_with_brake", "INST_BR PIN_PODNOSZENIE_03"
      (  in_safety_on                := "A-Flags".STATION.SAFETY_OK ,
         in_curtain_on               := "A-Flags".STATION.CURTAIN.OK ,
         in_move_hp                  := "A-DBVALVES".BR.PIN_RISING_03.in.move_hp ,
         in_move_wp                  := "A-DBVALVES".BR.PIN_RISING_03.in.move_wp ,
         in_move_idle                := "A-DBVALVES".BR.PIN_RISING_03.in.move_idle ,
         in_sensor_hp1               := I70.0 ,
         in_sensor_hp2               := I70.0 ,
         in_sensor_wp1               := I71.0 ,
         in_sensor_wp2               := I71.0 ,
         out_in_hp                   := "A-DBVALVES".BR.PIN_RISING_03.out.in_hp ,
         out_in_wp                   := "A-DBVALVES".BR.PIN_RISING_03.out.in_wp ,
         out_idle                    := "A-DBVALVES".BR.PIN_RISING_03.out.in_idle ,
         out_status                  := "A-DBVALVES".BR.PIN_RISING_03.out.status ,
         out_brake                   := #brake ,
         out_alarm_hp                := "A-DBVALVES".BR.PIN_RISING_03.out.alarm_hp ,
         out_alarm_wp                := "A-DBVALVES".BR.PIN_RISING_03.out.alarm_wp ,
         out_diag_status             := "A-DBVALVES".BR.PIN_RISING_03.out.diag_status ,
         in_ez_hp                    := Q3005.3 ,
         in_ez_wp                    := Q3005.2 ,
         in_ez_idle                  := "A-DBVALVES".BR.PIN_RISING_03.test.IDLE_DUMMY
      );

      CALL "3STATE_DIAG"
      (  in_diag_status              := "A-DBVALVES".BR.PIN_RISING_03.out.diag_status ,
         in_Ipw1                     := 'I70.0' ,
         in_Ipw2                     := ' ' ,
         in_Ipr1                     := 'I71.0' ,
         in_Ipr2                     := ' ' ,
         in_Qpw                      := 'Q3005.3' ,
         in_Qpr                      := 'Q3005.2' ,
         in_tio                      := "A-DBVALVES".io[9]
      );

      A "A-DBVALVES".BR.PIN_RISING_03.out.alarm_hp;
      = "A-ALARMS".VALVES.err0.%X14;

      A "A-DBVALVES".BR.PIN_RISING_03.out.alarm_wp;
      = "A-ALARMS".VALVES.err0.%X15;

      CALL "A-TESTSCL"
      (  in_nr                       := 9 ,
         out                         := "A-DBVALVES".BR.PIN_RISING_03.test
      );

      A(;
      L "A-Doku_DB_OP".HMI.Manual_Functions;
      L 9;
      <>I;
      );
      R "A-DBVALVES".BR.PIN_RISING_03.test.fp_HP;
      R "A-DBVALVES".BR.PIN_RISING_03.test.fp_WP;
      R "A-DBVALVES".BR.PIN_RISING_03.test.fp_IDLE;
NETWORK
TITLE = -

NETWORK
TITLE = [10] BR PIN_03 - HP
//[10] BR PIN_03 - HP
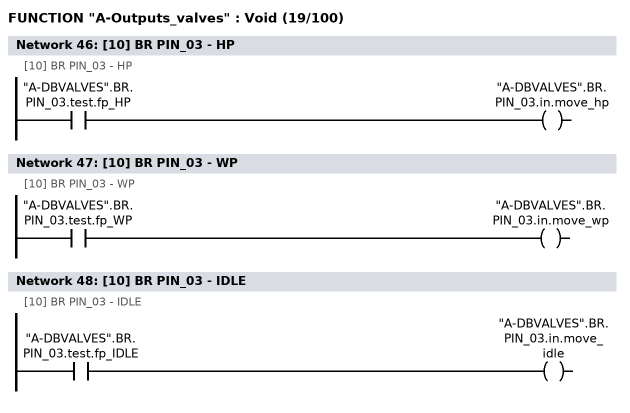
      O "A-DBVALVES".BR.PIN_03.test.fp_HP;
//    O     "A-Flags".STATION.IN_HP_STEP
      = "A-DBVALVES".BR.PIN_03.in.move_hp;
NETWORK
TITLE = [10] BR PIN_03 - WP
//[10] BR PIN_03 - WP
      O "A-DBVALVES".BR.PIN_03.test.fp_WP;
      = "A-DBVALVES".BR.PIN_03.in.move_wp;
NETWORK
TITLE = [10] BR PIN_03 - IDLE
//[10] BR PIN_03 - IDLE
      O "A-DBVALVES".BR.PIN_03.test.fp_IDLE;
      = "A-DBVALVES".BR.PIN_03.in.move_idle;
NETWORK
TITLE = [10] BR PIN_03
//[10] BR PIN_03
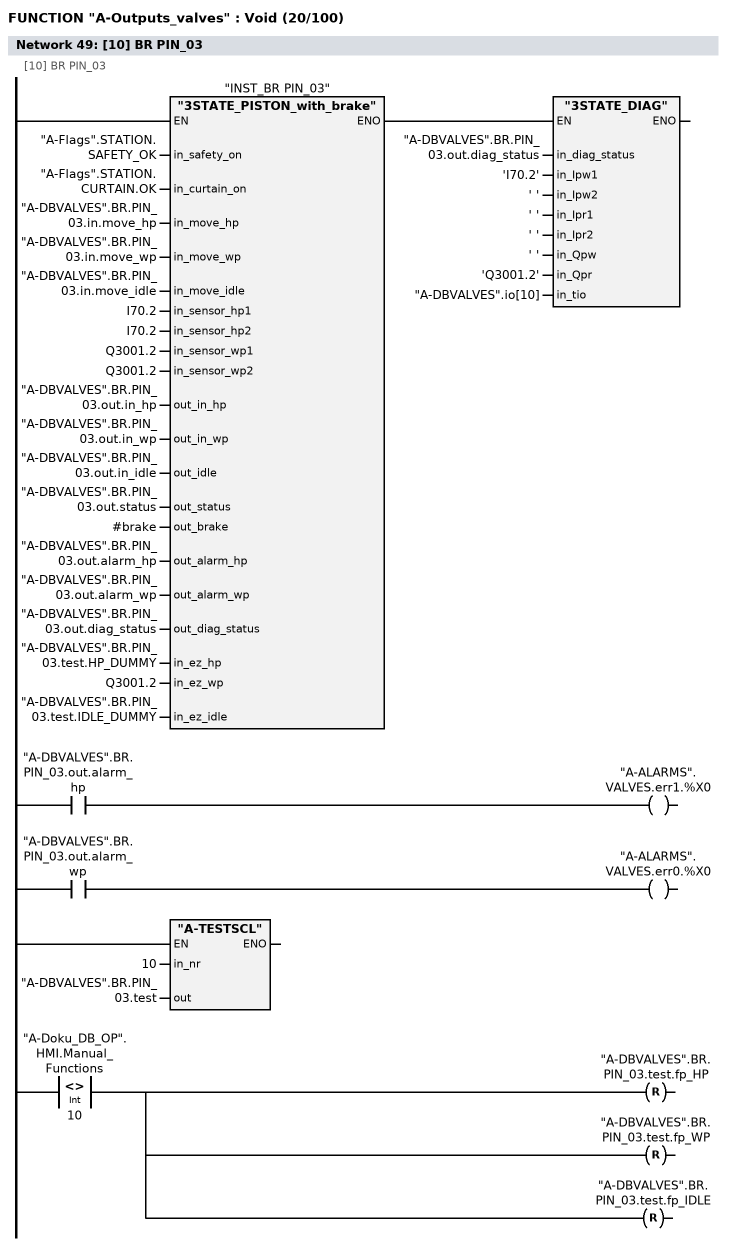
      CALL "3STATE_PISTON_with_brake", "INST_BR PIN_03"
      (  in_safety_on                := "A-Flags".STATION.SAFETY_OK ,
         in_curtain_on               := "A-Flags".STATION.CURTAIN.OK ,
         in_move_hp                  := "A-DBVALVES".BR.PIN_03.in.move_hp ,
         in_move_wp                  := "A-DBVALVES".BR.PIN_03.in.move_wp ,
         in_move_idle                := "A-DBVALVES".BR.PIN_03.in.move_idle ,
         in_sensor_hp1               := I70.2 ,
         in_sensor_hp2               := I70.2 ,
         in_sensor_wp1               := Q3001.2 ,
         in_sensor_wp2               := Q3001.2 ,
         out_in_hp                   := "A-DBVALVES".BR.PIN_03.out.in_hp ,
         out_in_wp                   := "A-DBVALVES".BR.PIN_03.out.in_wp ,
         out_idle                    := "A-DBVALVES".BR.PIN_03.out.in_idle ,
         out_status                  := "A-DBVALVES".BR.PIN_03.out.status ,
         out_brake                   := #brake ,
         out_alarm_hp                := "A-DBVALVES".BR.PIN_03.out.alarm_hp ,
         out_alarm_wp                := "A-DBVALVES".BR.PIN_03.out.alarm_wp ,
         out_diag_status             := "A-DBVALVES".BR.PIN_03.out.diag_status ,
         in_ez_hp                    := "A-DBVALVES".BR.PIN_03.test.HP_DUMMY ,
         in_ez_wp                    := Q3001.2 ,
         in_ez_idle                  := "A-DBVALVES".BR.PIN_03.test.IDLE_DUMMY
      );

      CALL "3STATE_DIAG"
      (  in_diag_status              := "A-DBVALVES".BR.PIN_03.out.diag_status ,
         in_Ipw1                     := 'I70.2' ,
         in_Ipw2                     := ' ' ,
         in_Ipr1                     := ' ' ,
         in_Ipr2                     := ' ' ,
         in_Qpw                      := ' ' ,
         in_Qpr                      := 'Q3001.2' ,
         in_tio                      := "A-DBVALVES".io[10]
      );

      A "A-DBVALVES".BR.PIN_03.out.alarm_hp;
      = "A-ALARMS".VALVES.err1.%X0;

      A "A-DBVALVES".BR.PIN_03.out.alarm_wp;
      = "A-ALARMS".VALVES.err0.%X0;

      CALL "A-TESTSCL"
      (  in_nr                       := 10 ,
         out                         := "A-DBVALVES".BR.PIN_03.test
      );

      A(;
      L "A-Doku_DB_OP".HMI.Manual_Functions;
      L 10;
      <>I;
      );
      R "A-DBVALVES".BR.PIN_03.test.fp_HP;
      R "A-DBVALVES".BR.PIN_03.test.fp_WP;
      R "A-DBVALVES".BR.PIN_03.test.fp_IDLE;
NETWORK
TITLE = -

NETWORK
TITLE = [11] BR PIN_PODNOSZENIE_04 - HP
//[11] BR PIN_RISING_04 - HP
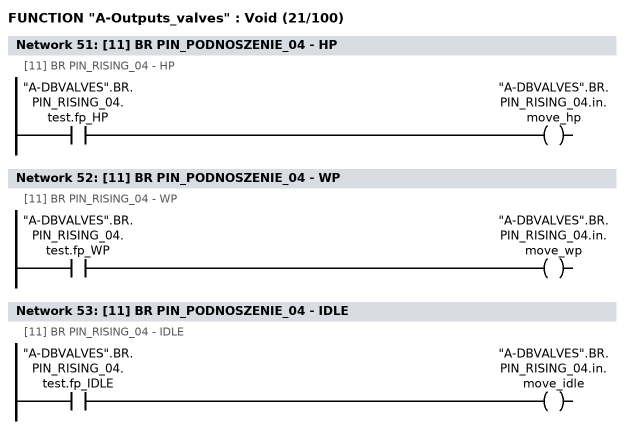
      O "A-DBVALVES".BR.PIN_RISING_04.test.fp_HP;
//    O     "A-Flags".STATION.IN_HP_STEP
      = "A-DBVALVES".BR.PIN_RISING_04.in.move_hp;
NETWORK
TITLE = [11] BR PIN_PODNOSZENIE_04 - WP
//[11] BR PIN_RISING_04 - WP
      O "A-DBVALVES".BR.PIN_RISING_04.test.fp_WP;
      = "A-DBVALVES".BR.PIN_RISING_04.in.move_wp;
NETWORK
TITLE = [11] BR PIN_PODNOSZENIE_04 - IDLE
//[11] BR PIN_RISING_04 - IDLE
      O "A-DBVALVES".BR.PIN_RISING_04.test.fp_IDLE;
      = "A-DBVALVES".BR.PIN_RISING_04.in.move_idle;
NETWORK
TITLE = [11] BR PIN_PODNOSZENIE_04
//[11] BR PIN_RISING_04
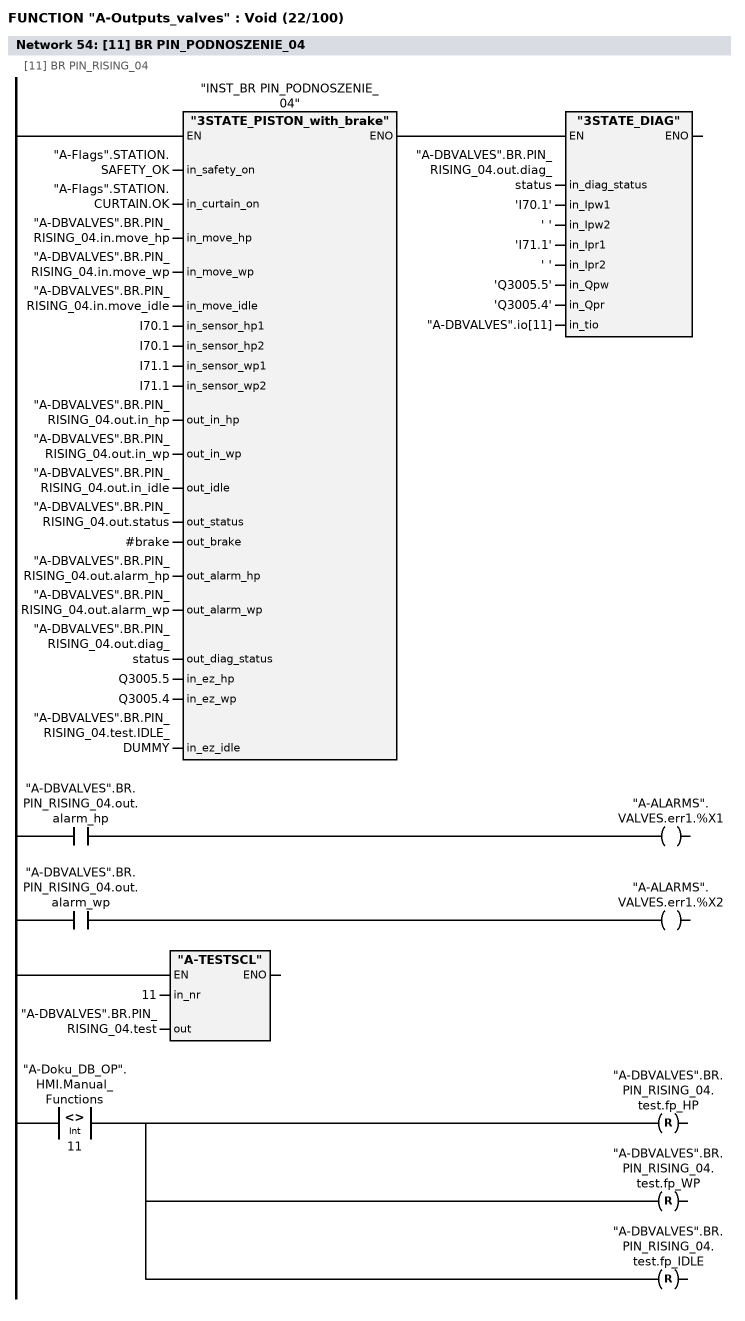
      CALL "3STATE_PISTON_with_brake", "INST_BR PIN_PODNOSZENIE_04"
      (  in_safety_on                := "A-Flags".STATION.SAFETY_OK ,
         in_curtain_on               := "A-Flags".STATION.CURTAIN.OK ,
         in_move_hp                  := "A-DBVALVES".BR.PIN_RISING_04.in.move_hp ,
         in_move_wp                  := "A-DBVALVES".BR.PIN_RISING_04.in.move_wp ,
         in_move_idle                := "A-DBVALVES".BR.PIN_RISING_04.in.move_idle ,
         in_sensor_hp1               := I70.1 ,
         in_sensor_hp2               := I70.1 ,
         in_sensor_wp1               := I71.1 ,
         in_sensor_wp2               := I71.1 ,
         out_in_hp                   := "A-DBVALVES".BR.PIN_RISING_04.out.in_hp ,
         out_in_wp                   := "A-DBVALVES".BR.PIN_RISING_04.out.in_wp ,
         out_idle                    := "A-DBVALVES".BR.PIN_RISING_04.out.in_idle ,
         out_status                  := "A-DBVALVES".BR.PIN_RISING_04.out.status ,
         out_brake                   := #brake ,
         out_alarm_hp                := "A-DBVALVES".BR.PIN_RISING_04.out.alarm_hp ,
         out_alarm_wp                := "A-DBVALVES".BR.PIN_RISING_04.out.alarm_wp ,
         out_diag_status             := "A-DBVALVES".BR.PIN_RISING_04.out.diag_status ,
         in_ez_hp                    := Q3005.5 ,
         in_ez_wp                    := Q3005.4 ,
         in_ez_idle                  := "A-DBVALVES".BR.PIN_RISING_04.test.IDLE_DUMMY
      );

      CALL "3STATE_DIAG"
      (  in_diag_status              := "A-DBVALVES".BR.PIN_RISING_04.out.diag_status ,
         in_Ipw1                     := 'I70.1' ,
         in_Ipw2                     := ' ' ,
         in_Ipr1                     := 'I71.1' ,
         in_Ipr2                     := ' ' ,
         in_Qpw                      := 'Q3005.5' ,
         in_Qpr                      := 'Q3005.4' ,
         in_tio                      := "A-DBVALVES".io[11]
      );

      A "A-DBVALVES".BR.PIN_RISING_04.out.alarm_hp;
      = "A-ALARMS".VALVES.err1.%X1;

      A "A-DBVALVES".BR.PIN_RISING_04.out.alarm_wp;
      = "A-ALARMS".VALVES.err1.%X2;

      CALL "A-TESTSCL"
      (  in_nr                       := 11 ,
         out                         := "A-DBVALVES".BR.PIN_RISING_04.test
      );

      A(;
      L "A-Doku_DB_OP".HMI.Manual_Functions;
      L 11;
      <>I;
      );
      R "A-DBVALVES".BR.PIN_RISING_04.test.fp_HP;
      R "A-DBVALVES".BR.PIN_RISING_04.test.fp_WP;
      R "A-DBVALVES".BR.PIN_RISING_04.test.fp_IDLE;
NETWORK
TITLE = -

NETWORK
TITLE = [12] BR PIN_04 - HP
//[12] BR PIN_04 - HP
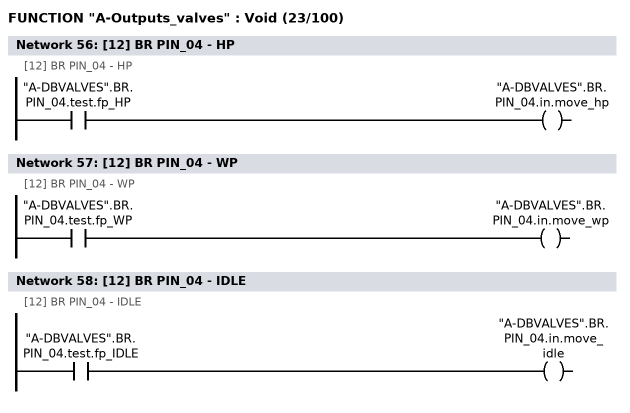
      O "A-DBVALVES".BR.PIN_04.test.fp_HP;
//    O     "A-Flags".STATION.IN_HP_STEP
      = "A-DBVALVES".BR.PIN_04.in.move_hp;
NETWORK
TITLE = [12] BR PIN_04 - WP
//[12] BR PIN_04 - WP
      O "A-DBVALVES".BR.PIN_04.test.fp_WP;
      = "A-DBVALVES".BR.PIN_04.in.move_wp;
NETWORK
TITLE = [12] BR PIN_04 - IDLE
//[12] BR PIN_04 - IDLE
      O "A-DBVALVES".BR.PIN_04.test.fp_IDLE;
      = "A-DBVALVES".BR.PIN_04.in.move_idle;
NETWORK
TITLE = [12] BR PIN_04
//[12] BR PIN_04
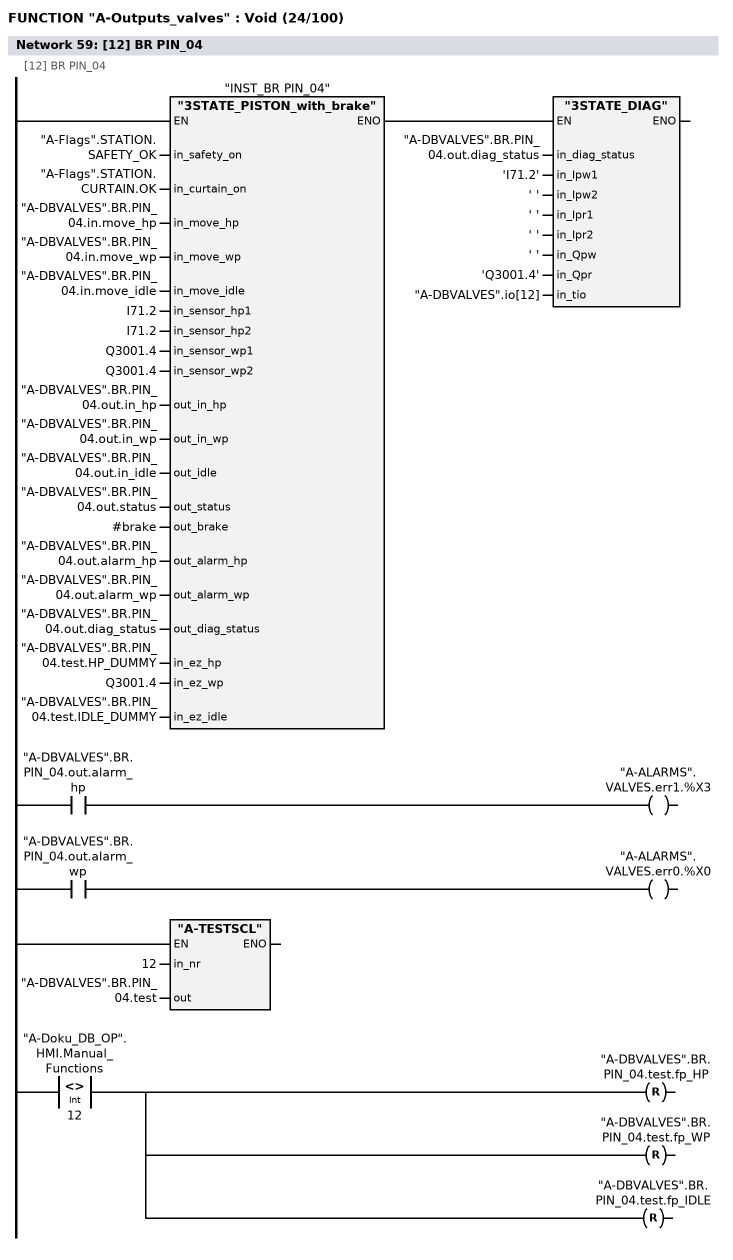
      CALL "3STATE_PISTON_with_brake", "INST_BR PIN_04"
      (  in_safety_on                := "A-Flags".STATION.SAFETY_OK ,
         in_curtain_on               := "A-Flags".STATION.CURTAIN.OK ,
         in_move_hp                  := "A-DBVALVES".BR.PIN_04.in.move_hp ,
         in_move_wp                  := "A-DBVALVES".BR.PIN_04.in.move_wp ,
         in_move_idle                := "A-DBVALVES".BR.PIN_04.in.move_idle ,
         in_sensor_hp1               := I71.2 ,
         in_sensor_hp2               := I71.2 ,
         in_sensor_wp1               := Q3001.4 ,
         in_sensor_wp2               := Q3001.4 ,
         out_in_hp                   := "A-DBVALVES".BR.PIN_04.out.in_hp ,
         out_in_wp                   := "A-DBVALVES".BR.PIN_04.out.in_wp ,
         out_idle                    := "A-DBVALVES".BR.PIN_04.out.in_idle ,
         out_status                  := "A-DBVALVES".BR.PIN_04.out.status ,
         out_brake                   := #brake ,
         out_alarm_hp                := "A-DBVALVES".BR.PIN_04.out.alarm_hp ,
         out_alarm_wp                := "A-DBVALVES".BR.PIN_04.out.alarm_wp ,
         out_diag_status             := "A-DBVALVES".BR.PIN_04.out.diag_status ,
         in_ez_hp                    := "A-DBVALVES".BR.PIN_04.test.HP_DUMMY ,
         in_ez_wp                    := Q3001.4 ,
         in_ez_idle                  := "A-DBVALVES".BR.PIN_04.test.IDLE_DUMMY
      );

      CALL "3STATE_DIAG"
      (  in_diag_status              := "A-DBVALVES".BR.PIN_04.out.diag_status ,
         in_Ipw1                     := 'I71.2' ,
         in_Ipw2                     := ' ' ,
         in_Ipr1                     := ' ' ,
         in_Ipr2                     := ' ' ,
         in_Qpw                      := ' ' ,
         in_Qpr                      := 'Q3001.4' ,
         in_tio                      := "A-DBVALVES".io[12]
      );

      A "A-DBVALVES".BR.PIN_04.out.alarm_hp;
      = "A-ALARMS".VALVES.err1.%X3;

      A "A-DBVALVES".BR.PIN_04.out.alarm_wp;
      = "A-ALARMS".VALVES.err0.%X0;

      CALL "A-TESTSCL"
      (  in_nr                       := 12 ,
         out                         := "A-DBVALVES".BR.PIN_04.test
      );

      A(;
      L "A-Doku_DB_OP".HMI.Manual_Functions;
      L 12;
      <>I;
      );
      R "A-DBVALVES".BR.PIN_04.test.fp_HP;
      R "A-DBVALVES".BR.PIN_04.test.fp_WP;
      R "A-DBVALVES".BR.PIN_04.test.fp_IDLE;
NETWORK
TITLE = -

NETWORK
TITLE = [13] BR BLAT5_PRZOD - HP
//[13] BR TABLE5_FRONT - HP
